// TwinCAT 3 PLC project xpp_pulsepicker_motion
// ProgramVersion: 3.1.4026.17
// libraries:
//   LCLS_OOPMotion, * (SLAC)
//   lcls_twincat_motion_synchronous, * (SLAC - LCLS)
//   PMPS, * (SLAC - LCLS)
//   Tc2_MC2, * (Beckhoff Automation GmbH)
//   Tc2_Standard, * (Beckhoff Automation GmbH)
//   Tc2_System, * (Beckhoff Automation GmbH)
//   TcUnit, * (www.tcunit.org)
// project tree:
//   DUTs/ E_ModeSelector.TcDUT, E_PickerState.TcDUT, E_StatusIndicator.TcDUT, E_ValidationStep.TcDUT, ST_SpeedProfile.TcDUT
//   / PlcTask.TcTTO
//   POUs/ FB_Burst.TcPOU, FB_FastClose.TcPOU, FB_FastOpen.TcPOU, FB_FlipFlop.TcPOU, FB_HomeToIndex.TcPOU, FB_MoveToNearestClosed.TcPOU, FB_OneShot.TcPOU, FB_PulsePicker.TcPOU, FB_SyncrhonousTest.TcPOU, MAIN.TcPOU
// real-time tasks:
//   TASK PlcTask: cycle T#1ms, priority 20, ADS port 350
// motion (NC):
//   TASK NC-Task 1 SAF: cycle T#1ms, priority 4, ADS port 501
//   TASK NC-Task 1 SVB: cycle T#10ms, priority 8, ADS port 511
//   AXIS Spindle (id 1)
//     General: UnitName=Degree
//     OtherSettings: AllowMotionCmdToSlave=true
//     encoder EncType=1
//     drive DrvType=5
//       Analog: TorqueSetpointScale=10, ScaleFactorActTorque=0.1
//       TimeComp: TaskDelayCycles=1
//     controller CtrType=1
//       CtrPara: PriorControlFactor=1
//         Observer: BandWidth=20
//   AXIS X (id 2)
//     OtherSettings: AllowMotionCmdToSlave=true
//     encoder EncType=1
//     drive DrvType=5
//       Analog: TorqueSetpointScale=10, ScaleFactorActTorque=0.1
//     controller CtrType=1
//       CtrPara: PriorControlFactor=1
//         Observer: BandWidth=20
//   AXIS Y (id 3)
//     OtherSettings: AllowMotionCmdToSlave=true
//     encoder EncType=1
//     drive DrvType=5
//       Analog: TorqueSetpointScale=10, ScaleFactorActTorque=0.1
//     controller CtrType=1
//       CtrPara: PriorControlFactor=1
//         Observer: BandWidth=20
// variable links:
//   xpp_pulsepicker_motion Instance <-> NC-Task 1 SAF/Axes/Spindle
//     PlcTask Inputs/MAIN.FB_SyncrhonousTest.AxisRef.NcToPlc <-> Outputs/ToPlc
//     PlcTask Outputs/MAIN.FB_SyncrhonousTest.AxisRef.PlcToNc <-> Inputs/FromPlc

CONFIGURATION xpp_pulsepicker_motion
    RESOURCE PLC ON TwinCAT3
        TASK PlcTask(INTERVAL := T#1ms, PRIORITY := 20);
        PROGRAM MAIN WITH PlcTask : MAIN;
    END_RESOURCE
END_CONFIGURATION

// ---- DUTs/E_ModeSelector.TcDUT
{attribute 'qualified_only'}
{attribute 'to_string'}
TYPE E_ModeSelector :
(
    ModeNone := 0,         // No mode / idle
    OneShot := 1,          // Mode 1
    FlipFlop := 2,         // Mode 2
    Burst := 3,            // Mode 3
    FastOpen := 4,         // Mode 4
    FastClose := 5,        // Mode 5
    Home := 7,             // Mode 7
    Reset := 99            // Reset
) UINT;
END_TYPE

// ---- DUTs/E_PickerState.TcDUT
{attribute 'qualified_only'}
{attribute 'strict'}
{attribute 'to_string'}
TYPE E_PickerState :
(
    Init,           // Startup: Read ModeSelect/SlitStatusFlag from NV
    HardReset,      // Hard reset initialization
    SoftReset,      // Soft reset/common block
    ModeSelect,     // Idle/waiting for user/command mode selection
    ModeExecute,    // Executing selected mode (One-Shot, Flip-Flop, etc)
    ErrorState      // Error or drift handling and recovery
);
END_TYPE

// ---- DUTs/E_StatusIndicator.TcDUT
{attribute 'qualified_only'}
{attribute 'strict'}
{attribute 'to_string'}
TYPE E_StatusIndicator :
(
// Mode Select/Resets
    WaitModeSelect := 0,
    // One-Shot
    OneShotInit := 10,
    OneShotLoopWait := 11,
    OneShotComplete := 12,
    // Flip-Flop
    FlipFlopInit := 20,
    FlipFlopLoopWait := 21,
    FlipFlopActive := 22,
    // Burst
    BurstInit := 30,
    BurstLoop := 31,
    // Fast Open/Close
    FastOpenInit := 40,
    FastOpenComplete := 41,
    FastCloseInit := 50,
    FastCloseComplete := 51,
    // Homing
    HomingInit := 70,
    HomingComplete := 79,
    // Special states
    HardReset := 80,
    SoftReset := 81
);
END_TYPE

// ---- DUTs/E_ValidationStep.TcDUT
{attribute 'qualified_only'}
{attribute 'strict'}
{attribute 'to_string'}
TYPE E_ValidationStep :
(
	INITIALIZE := 0,
	WAIT_FOR_IDLE,
	COMMAND_SEQUENCE_START,
	GENERATE_TARGET_POINTS,
	COMMAND_MOVE_TO_FIRST_TARGET,
	COMMAND_START_TRIGGERS,
	CONFIRM_BACK_TO_IDLE
);
END_TYPE

// ---- DUTs/ST_SpeedProfile.TcDUT
TYPE ST_SpeedProfile :
STRUCT
	InitialVelocity : LREAL;
	MaxVelocity : LREAL;
	Acceleration : LREAL;
	Deceleration : LREAL;
END_STRUCT
END_TYPE

// ---- POUs/MAIN.TcPOU
PROGRAM MAIN
VAR
	FB_SyncrhonousTest : FB_SyncrhonousTest;
END_VAR

FB_SyncrhonousTest();

END_PROGRAM

// ---- POUs/FB_SyncrhonousTest.TcPOU
FUNCTION_BLOCK FB_SyncrhonousTest
VAR
    (* --- Axis Reference --- *)
    AxisRef : AXIS_REF;

	fbPersistentDataStorage : FB_PersistentDataStorage;
    fbMotionStage : FB_MotionStageNC(
        sName := 'Test2',
         AxisRef := AxisRef,
        iPersistentDataStorage := fbPersistentDataStorage
    ) := (HomeMode:=E_EpicsHomeCmd.LOW_LIMIT);
	
    (* --- Timing, Trigger, and Clock --- *)
//     fbClockSourceInternal    : FB_ClockSourceInternal(
//         nTimePerScan := 250000,            // 0.25 ms cycle
//         nStartingTime := 0
//     );
    fbClockSourceInternal    : FB_ClockSourceInternal(
        nTimePerScan := 1000000,            // 1 ms cycle
        nStartingTime := 0
    );	
 	fbClockSourceEtherCATDistributedClock : FB_ClockSourceEtherCATDistributedClock;
//     fbTriggerSourceInternal : FB_TriggerSourceInternal(
//         iClockSource := fbClockSourceEtherCATDistributedClock
//     );
    fbTriggerSourceInternal : FB_TriggerSourceInternal(
        iClockSource := fbClockSourceEtherCATDistributedClock
    );
	
    fbTriggerManagerInternal : FB_TriggerManager(
        fTriggerFrequencyExpected := 30.0,  // 30 Hz expected trigger input
        iTriggerSource := fbTriggerSourceInternal
    );
//     fbTrajectoryClockSynchronous: FB_TrajectoryClockSynchronous (
//         fCycleTime := 0.000250,
//         iClockSource := fbClockSourceEtherCATDistributedClock
//     );
//     fbTrajectoryClockSynchronous: FB_TrajectoryClockSynchronous (
//         fCycleTime := 0.000250,
//         iClockSource := fbClockSourceInternal
//     );
    fbTrajectoryClockSynchronous: FB_TrajectoryClockSynchronous (
        fCycleTime := 0.001,
        iClockSource := fbClockSourceInternal
    );
    (* --- Trajectory and Buffer --- *)
    fbTargetPointSynchronousQueue        : FB_TargetPointSynchronousQueue<6>;   // Buffer of size 6
    fbTargetPointSynchronousLoader     		 : FB_TargetPointSynchronousLoaderFromEpics<1,6>(
        nMaxNumPointsProcessedPerCycle := 10
    );

    (* --- Setpoint & Feedback Interfaces --- *)
    fbSetpointInterfaceNC  : FB_SetpointInterfaceNC(AxisRef := AxisRef);
    fbFeedbackInterfaceNC  : FB_FeedbackInterfaceNC(AxisRef := AxisRef);

    (* --- Trajectory Synchronous and Error Estimation --- *)
    fbTrajectorySynchronous : FB_TrajectorySynchronousBezierContinuousSnap(
        iTrajectoryClock := fbTrajectoryClockSynchronous,
		bCalcPosPoints := TRUE,
		bCalcVelPoints := TRUE,
		bCalcAccPoints := TRUE,
		bCalcJerkPoints := TRUE,
		bCalcSnapPoints := TRUE
    );
    fbErrorEstimator     : FB_ErrorEstimator(
        iTrajectoryClock := fbTrajectoryClockSynchronous,
        iFeedbackInterface := fbFeedbackInterfaceNC,
        iTargetPointSynchronousQueue := fbTargetPointSynchronousQueue,
        iTrajectorySynchronous := fbTrajectorySynchronous,
        iTriggerManager := fbTriggerManagerInternal
    );

    (* --- Setpoint Generator --- *)
    fbSetpointGeneratorContinuousSynchronous : FB_SetpointGeneratorContinuousSynchronous(
        fTimeSyncGain := 0.2,
		iSetpointInterface := fbSetpointInterfaceNC,
		iFeedbackInterface := fbFeedbackInterfaceNC,
		iErrorEstimator := fbErrorEstimator,
		iTrajectorySynchronous := fbTrajectorySynchronous,
		iTargetPointSynchronousQueue := fbTargetPointSynchronousQueue,
		iTrajectoryClock := fbTrajectoryClockSynchronous,
		iTriggerManager := fbTriggerManagerInternal
    );

    (* --- Sequencer and EPICS Command/Loader --- *)
    fbTrajectorySequencerCommandsFromEpics : FB_TrajectorySequencerCommandsFromEpics;
	
    fbTrajectorySequencerSynchronous : FB_TrajectorySequencerSynchronous<1>(
        iTriggerManager := fbTriggerManagerInternal,
        iTrajectorySequencerCommands := fbTrajectorySequencerCommandsFromEpics
    );

	arTrajectoryPositions : ARRAY[1..6] OF LREAL := [
		-11.25,   // up: start
		-6.11,    // up: end / down: start
		-0.33,    // down: end / flat: start
		 0.33,    // flat: end / ramp2: start
		 6.12,    // ramp2: end / final: start
		11.25     // final: end
	];
	
	arTargetVelocities : ARRAY[1..6] OF LREAL := [
		 0.0,     // up: start
	  2400.0,     // up: end / down: start
	   300.0,     // down: end / flat: start
	   300.0,     // flat: end / ramp2: start
	  2400.0,     // ramp2: end / final: start
		 0.0      // final: end
	];
	
	arTargetTime : ARRAY[1..6] OF LREAL := [
	  0.0,            // up: start
	  0.0042828125,   // up: end / down: start
	  0.008565625,    // down: end / flat: start
	  0.010765625,    // flat: end / ramp2: start
	  0.0150484375,   // ramp2: end / final: start
	  0.01933125      // final: end
	];
    stPoint : ST_TrajectorySynchronousPoint;
	fbTargetPointSynchronous : FB_TargetPointSynchronous;
	bHardwareEnableSync AT %Q* :  BOOL;
	i : INT;
    (* --- Optionally: index/scan flags, and utility vars for test harness --- *)
    firstScan  : BOOL := TRUE;
    nIndex     : INT  := 1;         // Not needed for single axis, just in case
    seqStep    : E_TrajectorySequenceStep;
    isIdle     : BOOL;
	eUserState : E_ValidationStep;
	bHome: BOOL;
	bStartCommand: BOOL;
	bCommandMoveToFirstTarget: BOOL;
	bQuitEarly: BOOL;
	bStartTriggers: BOOL;
END_VAR

IF firstScan THEN

	bHardwareEnableSync := TRUE;
	fbMotionStage.EnableMode := LCLS_OOPMotion.E_StageEnableMode.ALWAYS;
	fbMotionStage.MotionCmd.nCmdData := LCLS_OOPMotion.E_EpicsHomeCmd.LOW_LIMIT;
	fbMotionStage.MotionCmd.fVelocity:=12.5;
	fbMotionStage.MotionCmd.fDeceleration := 25.5;
	fbMotionStage.MotionCmd.fAcceleration:=25.5;
	fbMotionStage.MotionCmd.fHomePosition := 0;

//     fbTriggerSource.Start(
//         fFrequency := 30.0,
//         nTotalNumTriggers := 1
//     );
// 	
//     fbTriggerSource.Reset();
//     fbTrajectorySequencerSynchronous.Register(
//         iTargetPointSynchronousQueue := fbTargetPointSynchronousQueue,
//         iSetpointGeneratorContinuous := fbSetpointGen,
//         iMotionStage := fbMotionStage,            // Use the motion axis FB here!
//         iSetpointInterface := fbSetpointInterface
//     );
    firstScan := FALSE;
END_IF

IF bHome THEN
	fbMotionStage.MotionCmd.bHomeCmd := TRUE;
	bHome := FALSE;
END_IF

fbClockSourceInternal();
//fbClockSourceEtherCATDistributedClock();
fbTriggerSourceInternal();
fbTrajectoryClockSynchronous();
fbTriggerManagerInternal();

// call for each axis
fbMotionStage();

fbSetpointInterfaceNC();
fbErrorEstimator();
fbSetpointGeneratorContinuousSynchronous();
fbTrajectorySequencerSynchronous();
///////////////////////////////////
fbTrajectorySequencerSynchronous();

CASE eUserState OF
	E_ValidationStep.INITIALIZE:
	 	fbTriggerSourceInternal.Reset();
        //fbTriggerManager.ResetTriggerCounter();
        fbTriggerManagerInternal.ResetTriggerCounter();
		
		fbTrajectorySequencerSynchronous.Register(
			iTargetPointSynchronousQueue := fbTargetPointSynchronousQueue,
			iSetpointGeneratorContinuous := fbSetpointGeneratorContinuousSynchronous,
			iMotionStage := fbMotionStage,            // Use the motion axis FB here!
			iSetpointInterface := fbSetpointInterfaceNC
		);
		eUserState := E_ValidationStep.WAIT_FOR_IDLE;
		
    E_ValidationStep.WAIT_FOR_IDLE:
        IF fbTrajectorySequencerSynchronous.eSequenceStep = E_TrajectorySequenceStep.IDLE THEN
            eUserState := E_ValidationStep.COMMAND_SEQUENCE_START;
        END_IF
		
    E_ValidationStep.COMMAND_SEQUENCE_START:
		IF bStartCommand THEN
			fbTrajectorySequencerCommandsFromEpics.CommandSequenceStart := TRUE;
		
			eUserState := E_ValidationStep.GENERATE_TARGET_POINTS;
			
			bStartCommand := FALSE;
		END_IF
	E_ValidationStep.GENERATE_TARGET_POINTS:
		FOR i := 1 TO 6 DO
			fbTargetPointSynchronous.Position := arTrajectoryPositions[i];
			fbTargetPointSynchronous.T := arTargetTime[i];
	
			fbTargetPointSynchronous.Velocity := arTargetVelocities[i];   // If your system uses velocity (optional)
			fbTargetPointSynchronous.Acceleration := 0.0;
			fbTargetPointSynchronous.Jerk := 0.0;
			fbTargetPointSynchronous.Snap := 0.0;
			fbTargetPointSynchronousQueue.Push(fbTargetPointSynchronous);
		END_FOR
		eUserState := E_ValidationStep.COMMAND_MOVE_TO_FIRST_TARGET;
		
    E_ValidationStep.COMMAND_MOVE_TO_FIRST_TARGET:
        IF bCommandMoveToFirstTarget THEN
            fbTrajectorySequencerCommandsFromEpics.CommandSequenceMoveToFirstTarget := TRUE;

            eUserState := E_ValidationStep.COMMAND_START_TRIGGERS;
			
			bCommandMoveToFirstTarget := FALSE;
        ELSIF fbTrajectorySequencerSynchronous.eSequenceStep = E_TrajectorySequenceStep.CONF_ERROR_RESET THEN
            bQuitEarly := TRUE;
        END_IF
		
    E_ValidationStep.COMMAND_START_TRIGGERS:
        IF bStartTriggers THEN
            //fbTriggerSourceInternal.Start(fFrequency := GVL_Constants.fTargetFrequency, nTotalNumTriggers := nNumTargets);
			fbTriggerSourceInternal.Start(
				fFrequency := 30.0,
				nTotalNumTriggers := 1
			);
            eUserState := E_ValidationStep.CONFIRM_BACK_TO_IDLE;
			
			bStartTriggers := FALSE;
        ELSIF fbTrajectorySequencerSynchronous.eSequenceStep = E_TrajectorySequenceStep.CONF_ERROR_RESET THEN
            bQuitEarly := TRUE;
        END_IF
		
	E_ValidationStep.CONFIRM_BACK_TO_IDLE:
        IF fbTrajectorySequencerSynchronous.eSequenceStep = E_TrajectorySequenceStep.IDLE THEN
            eUserState := E_ValidationStep.COMMAND_SEQUENCE_START;
        ELSIF fbTrajectorySequencerSynchronous.eSequenceStep = E_TrajectorySequenceStep.CONF_ERROR_RESET THEN
            bQuitEarly := TRUE;
        END_IF
END_CASE

END_FUNCTION_BLOCK

// ---- POUs/FB_Burst.TcPOU
FUNCTION_BLOCK FB_Burst
VAR_INPUT
    MotorCenterPosition : INT;              // P0
    MotorClosedPositionPlus : INT;          // P1
    EncoderCenterPosition : INT;            // N0
    EncoderClosedPositionPlus : INT;        // N1
    DriftLimit : INT;                       // Dl
    ErrorCheckEnabled : BOOL;               // Ec
    C2 : INT;                               // Actual encoder count
    InputTrip : BOOL;                       // Rising edge is Input trigger
END_VAR
VAR_IN_OUT
    EncoderShadow : INT;                    // Cs (shadow reg)
    SlitStatusFlag : INT;                   // Df
    UpperDriftViolations : INT;             // Ud
    LowerDriftViolations : INT;             // Ld
END_VAR
VAR_OUTPUT
    Complete : BOOL := FALSE;               // Set TRUE when any move is complete
END_VAR
VAR
    State : INT := 0;                       // 0=idle, 1=open move, 2=close move, 10=waiting for input
    Drift : INT := 0;
    InputTripLast : BOOL := FALSE;          // For edge detection
END_VAR

METHOD Execute
// Edge detection
VAR
    Trip : BOOL;
END_VAR
Trip := InputTrip AND NOT InputTripLast;
InputTripLast := InputTrip;

// Main burst loop. User triggers with input pulse.
// Initial state: waiting for InputTrip, Df determines direction
IF State = 0 THEN
    IF Trip THEN
        IF SlitStatusFlag = 1 THEN     // Currently closed, need to open on trip
            StartOpenMove();
        ELSE                           // Currently open, need to close on trip
            StartCloseMove();
        END_IF
    END_IF
ELSIF State = 1 THEN
    // J3: Burst Open ISR
    // Move shutter to open position (MotorCenterPosition)
    // Replace with MC_MoveAbsolute or actual axis block (simulate instant success here)
    IF ErrorCheckEnabled AND (SlitStatusFlag = 1) THEN
        Drift := EncoderClosedPositionPlus - EncoderShadow; // N1-Cs
        IF Drift >= DriftLimit THEN
            LowerDriftViolations := LowerDriftViolations + 1;
        END_IF
    END_IF
    EncoderShadow := C2;
    SlitStatusFlag := 0;   // Slits are open
    State := 10;           // Waiting for next input pulse
    Complete := TRUE;

ELSIF State = 2 THEN
    // J4: Burst Close ISR
    // Move shutter to closed position (MotorClosedPositionPlus)
    // Replace with MC_MoveAbsolute or actual axis block (simulate instant success here)
    IF ErrorCheckEnabled THEN
        Drift := EncoderShadow - EncoderCenterPosition; // Cs-N0
        IF Drift >= DriftLimit THEN
            UpperDriftViolations := UpperDriftViolations + 1;
        END_IF
    END_IF
    EncoderShadow := C2;
    SlitStatusFlag := 1;   // Slits are closed
    State := 10;           // Waiting for next input pulse
    Complete := TRUE;

ELSIF State = 10 THEN
    // Await next trigger
    IF Trip THEN
        IF SlitStatusFlag = 1 THEN
            StartOpenMove();
        ELSE
            StartCloseMove();
        END_IF
    END_IF
END_IF
END_METHOD

METHOD StartCloseMove
VAR_INPUT
END_VAR
    State := 2;          // Start close move ISR (J4)
    Complete := FALSE;
END_METHOD

METHOD StartOpenMove
VAR_INPUT
END_VAR
    State := 1;          // Start open move ISR (J3)
    Complete := FALSE;
END_METHOD

END_FUNCTION_BLOCK

// ---- POUs/FB_FastClose.TcPOU
FUNCTION_BLOCK FB_FastClose
VAR_INPUT
    MotorClosedPositionPlus : INT;       // P1 (positive closed)
    C2 : INT;                            // Encoder actual count
    SlitStatusFlagIn : INT;              // Input Df for position check
END_VAR
VAR_IN_OUT
    EncoderShadow : INT;                 // Cs (shadow register)
    SlitStatusFlag : INT;                // Df
END_VAR
VAR_OUTPUT
    Complete : BOOL := FALSE;
END_VAR
VAR
    State : INT := 0; // 0: idle, 1: moving, 2: done
END_VAR

METHOD Execute : BOOL
VAR_INPUT
END_VAR
IF State = 0 THEN
    // Only move if not already closed
    IF (SlitStatusFlagIn <> 1) AND (SlitStatusFlagIn <> -1) THEN
        State := 1;       // Start moving to P1
        Complete := FALSE;
    ELSE
        // Already closed, skip to complete
        State := 2;
        Complete := TRUE;
    END_IF
ELSIF State = 1 THEN
    // Simulate motion complete; check actual axis in a real system
    EncoderShadow := C2;
    SlitStatusFlag := 1;   // Positive closed
    State := 2;
    Complete := TRUE;
END_IF
END_METHOD

METHOD Reset : BOOL
VAR_INPUT
END_VAR
    State := 0;
    Complete := FALSE;
END_METHOD

END_FUNCTION_BLOCK

// ---- POUs/FB_FastOpen.TcPOU
FUNCTION_BLOCK  FB_FastOpen
VAR_INPUT
    MotorCenterPosition : INT;           // P0 (open pos)
    C2 : INT;                            // Encoder actual count
END_VAR
VAR_IN_OUT
    EncoderShadow : INT;                 // Cs (shadow register)
    SlitStatusFlag : INT;                // Df
END_VAR
VAR_OUTPUT
    Complete : BOOL := FALSE;
END_VAR
VAR
    State : INT := 0; // 0: idle, 1: moving, 2: done
END_VAR

METHOD Execute : BOOL
VAR_INPUT
END_VAR
IF State = 0 THEN
    // Start movement to open (simulate instant success; call MC_MoveAbsolute in real system)
    State := 1;
    Complete := FALSE;
ELSIF State = 1 THEN
    // Simulate motion complete; check actual motion in real system
    EncoderShadow := C2;
    SlitStatusFlag := 0;      // Open
    State := 2;
    Complete := TRUE;
END_IF
END_METHOD

METHOD Reset : BOOL
VAR_INPUT
END_VAR
    State := 0;
    Complete := FALSE;
END_METHOD

END_FUNCTION_BLOCK

// ---- POUs/FB_FlipFlop.TcPOU
FUNCTION_BLOCK FB_FlipFlop
VAR_INPUT
    MotorClosedPositionPlus  : INT;            // P1
    MotorClosedPositionMinus : INT;            // P2
    EncoderClosedPositionPlus: INT;            // N1
    EncoderClosedPositionMinus: INT;           // N2
    DriftLimit               : INT;
    ErrorCheckEnabled        : BOOL;
    C2                       : INT;            // encoder count
    InputTrip                : BOOL;           // TRUE on input pulse
END_VAR
VAR_IN_OUT
    EncoderShadow            : INT;            // Cs
    SlitStatusFlag           : INT;            // Df
    UpperDriftViolations     : INT;            // Ud
    LowerDriftViolations     : INT;            // Ld
END_VAR
VAR_OUTPUT
    Complete                 : BOOL := FALSE;  // TRUE when first move done
END_VAR
VAR
    NextDirectionPos         : BOOL := TRUE;   // TRUE: Arm ISR2/J6, FALSE: Arm ISR1/J5
    State                    : INT := 0;       // 0: idle/init; 1: closed pos armed; 2: waiting trip; 3: actuation/move
    LastInputTrip            : BOOL := FALSE;  // For edge detection
    Drift                    : INT := 0;
END_VAR

METHOD Execute : BOOL
VAR
    Trip : BOOL;
END_VAR
Trip := InputTrip AND NOT LastInputTrip;
LastInputTrip := InputTrip;

// Init: ensure we're at positive or negative closed
IF State=0 THEN
    IF (SlitStatusFlag = -1) THEN
        NextDirectionPos := TRUE;  // Arm ISR2/J6 on trip
    ELSE
        NextDirectionPos := FALSE; // Arm ISR1/J5 on trip
    END_IF
    State := 1;
    Complete := TRUE;              // First move is done on entry
ELSIF State=1 OR State=2 THEN
    // Wait for input trip
    IF Trip THEN
        State := 3;
        Complete := FALSE;
    END_IF
ELSIF State=3 THEN
    // Do move and drift calculation
    IF NextDirectionPos THEN
        // ISR2/J6: P2→P1
        // Move motor to P1 (simulate instant for demo)
        IF ErrorCheckEnabled THEN
            Drift := EncoderShadow - EncoderClosedPositionMinus; // Cs-N2
            IF Drift >= DriftLimit THEN
                UpperDriftViolations := UpperDriftViolations + 1;
            END_IF
        END_IF
        SlitStatusFlag := 1;    // Positive closed
        EncoderShadow := C2;
        NextDirectionPos := FALSE; // Next trip arms negative direction (J5)
    ELSE
        // ISR1/J5: P1→P2
        // Move motor to P2 (simulate instant for demo)
        IF ErrorCheckEnabled THEN
            Drift := EncoderClosedPositionPlus - EncoderShadow; // N1-Cs
            IF Drift >= DriftLimit THEN
                LowerDriftViolations := LowerDriftViolations + 1;
            END_IF
        END_IF
        SlitStatusFlag := -1;   // Negative closed
        EncoderShadow := C2;
        NextDirectionPos := TRUE; // Next trip arms positive direction (J6)
    END_IF
    State := 2;    // Return to wait for input trip
    Complete := TRUE;
END_IF
END_METHOD

METHOD Reset : BOOL
VAR_INPUT
END_VAR
    State := 0;
    Complete := FALSE;
    NextDirectionPos := TRUE; // Default to J6
END_METHOD

END_FUNCTION_BLOCK

// ---- POUs/FB_HomeToIndex.TcPOU
FUNCTION_BLOCK FB_HomeToIndex
VAR_INPUT
    MotorClosedPositionPlus : INT;   // P1
    EncoderClosedPositionPlus: INT;  // N1
    MagicOffset : INT;               // Mo
    HomingSpeed : LREAL;      // CL V9 (see earlier struct)
    VM : LREAL;                        // Max velocity (from speed profile)
END_VAR
VAR_IN_OUT
    EncoderShadow : INT;             // Cs
    SlitStatusFlag : INT;            // Df
    Ud : INT;                        // Upper drift violation counter
    Lowerd : INT;                        // Lower drift violation counter
END_VAR
VAR_OUTPUT
    Complete : BOOL := FALSE;
END_VAR
VAR
    State : INT := 0;
    DoneHome : BOOL := FALSE;
    DoneOffset : BOOL := FALSE;
END_VAR

METHOD Execute : BOOL
VAR_INPUT
END_VAR
// State 0: Start Homing
IF State = 0 THEN
    // Load homing speed profile (CL V9) - can set to axis FB
    // (Your MC_Home or similar FB called here with VM etc.)
    // For demo, just set DoneHome true immediately, replace with real move!
    DoneHome := TRUE;
    State := 1;
END_IF

// State 1: Wait for Homing move complete
IF State = 1 THEN
    IF DoneHome THEN
        // Now do relative move by magic offset to positive closed (P1)
        // MC_MoveRelative(Mo ...) here in real system!
        DoneOffset := TRUE;
        State := 2;
    END_IF
END_IF

// State 2: Wait for move by Mo complete
IF State = 2 THEN
    IF DoneOffset THEN
        // Set C1 and C2 appropriately
        // In real code, set axis reference to MotorClosedPositionPlus
        // Set encoder reference to EncoderClosedPositionPlus
        // Sync shadow register
        // Set slit state Df to known positive closed
        SlitStatusFlag := 1;
        EncoderShadow := EncoderClosedPositionPlus;
        Ud := 0;
        Lowerd := 0;
        Complete := TRUE;
        State := 3;
    END_IF
END_IF
END_METHOD

METHOD Reset : BOOL
VAR_INPUT
END_VAR
    State := 0;
    DoneHome := FALSE;
    DoneOffset := FALSE;
    Complete := FALSE;
END_METHOD

END_FUNCTION_BLOCK

// ---- POUs/FB_MoveToNearestClosed.TcPOU
FUNCTION_BLOCK FB_MoveToNearestClosed
VAR_INPUT
    MotorClosedPositionPlus : INT;    // P1
    C2 : INT;                         // Actual encoder count (from axis/encoder)
    SlitStatusFlagIn : INT;           // Input Df (current position status)
END_VAR
VAR_IN_OUT
    EncoderShadow : INT;              // Cs, shadow register for drift checking
    SlitStatusFlag : INT;             // Df, output position status
END_VAR
VAR_OUTPUT
    Complete : BOOL := FALSE;
END_VAR
VAR
    State : INT := 0;                 // 0: ready, 1: moving, 2: done
END_VAR

METHOD Execute : BOOL
VAR_INPUT
END_VAR
IF State = 0 THEN
    IF (SlitStatusFlagIn <> 1) AND (SlitStatusFlagIn <> -1) THEN
        // Start the move to P1 (simulate or call MC_MoveAbsolute)
        State := 1;
        Complete := FALSE;
    ELSE
        // Already closed; nothing to do
        State := 2;
        Complete := TRUE;
    END_IF
ELSIF State = 1 THEN
    // Simulate move complete; in real code, check axis feedback!
    EncoderShadow := C2;
    SlitStatusFlag := 1;         // Signal at positive closed position
    State := 2;
    Complete := TRUE;
END_IF
END_METHOD

METHOD Reset : BOOL
VAR_INPUT
END_VAR
    State := 0;
    Complete := FALSE;
END_METHOD

END_FUNCTION_BLOCK

// ---- POUs/FB_OneShot.TcPOU
FUNCTION_BLOCK FB_OneShot
VAR_INPUT
    MotorClosedPositionPlus : INT;        // P1
    MotorClosedPositionMinus : INT;       // P2
    EncoderClosedPositionPlus : INT;      // N1
    EncoderClosedPositionMinus : INT;     // N2
    DriftLimit : INT;                     // Dl
    ErrorCheckEnabled : BOOL;             // Ec
    C2 : INT;                             // Actual encoder count
    ArmDirectionPos : BOOL := TRUE;       // TRUE: arm ISR2/P2→P1, FALSE: arm ISR1/P1→P2
    TriggerInputTrip : BOOL;              // TRUE when Input Trip triggers the action
END_VAR
VAR_IN_OUT
    EncoderShadow : INT;                  // Cs
    SlitStatusFlag : INT;                 // Df
    UpperDriftViolations : INT;           // Ud
    LowerDriftViolations : INT;           // Ld
END_VAR
VAR_OUTPUT
    Complete : BOOL := FALSE;             // Set TRUE when done
END_VAR
VAR
    Drift : INT := 0;
    MotionState : INT := 0;               // 0: idle/armed, 1: running, 2: done
END_VAR

METHOD Execute : BOOL
VAR_INPUT
END_VAR
// Call cyclically while armed; runs the ISR sequence after Input Trip
IF MotionState = 0 THEN
    // Nothing until InputTrip triggers
    IF TriggerInputTrip THEN
        MotionState := 1;         // Begin movement
        Complete := FALSE;
    END_IF
ELSIF MotionState = 1 THEN
    // Axis move (simulate or use your axis FB)
    IF ArmDirectionPos THEN
        // Move P2=>P1 (positive)
        // Example: AxisControl.MoveAbs(MotorClosedPositionPlus) -- Replace with FB or IO
        // Simulate motion complete immediately for demo!
        IF ErrorCheckEnabled THEN
            Drift := EncoderShadow - EncoderClosedPositionMinus; // Dr = Cs - N2
            IF Drift >= DriftLimit THEN
                UpperDriftViolations := UpperDriftViolations + 1;
            END_IF
        END_IF
        SlitStatusFlag := 1;     // Positive closed
    ELSE
        // Move P1=>P2 (negative)
        // Example: AxisControl.MoveAbs(MotorClosedPositionMinus)
        IF ErrorCheckEnabled THEN
            Drift := EncoderClosedPositionPlus - EncoderShadow; // Dr = N1 - Cs
            IF Drift >= DriftLimit THEN
                LowerDriftViolations := LowerDriftViolations + 1;
            END_IF
        END_IF
        SlitStatusFlag := -1;    // Negative closed
    END_IF
    EncoderShadow := C2;
    MotionState := 2;             // Finished
    Complete := TRUE;
END_IF
END_METHOD

METHOD Reset : BOOL
VAR_INPUT
END_VAR
    MotionState := 0;
    Complete := FALSE;
END_METHOD

END_FUNCTION_BLOCK

// ---- POUs/FB_PulsePicker.TcPOU
FUNCTION_BLOCK FB_PulsePicker
VAR PERSISTENT
    ModeSelect : E_ModeSelector := E_ModeSelector.ModeNone;;
 	StatusIndicator : E_StatusIndicator := E_StatusIndicator.WaitModeSelect;
    SlitStatusFlag : INT := 99;
    SweepDistance : INT;      
    EncoderSweepDistance : INT;
    EncoderDrift : INT;
    DriftLimit : INT;
    MotorCenterPosition : INT;
    MotorClosedPositionPlus : INT;    // P1
    MotorClosedPositionMinus : INT;   // P2
    EncoderCenterPosition : INT;      // N0
    EncoderClosedPositionPlus : INT;  // N1
    EncoderClosedPositionMinus : INT; // N2
    ErrorCheckEnabled : BOOL;
    MCodeVersion : INT;
    HeartbeatCounter : INT;
    EncoderShadow : INT;              // Cs
    UpperDriftViolations : INT;       // Ud
    LowerDriftViolations : INT;       // Ld
    HomingOffset : INT;               // Mo

END_VAR

VAR
    CurrentState : E_PickerState := E_PickerState.Init;
    ErrorCode : INT := 0;
    UserModeReq : UINT := 0;       // From HMI or remote
    (* Axis/encoder for simulation *)
    C2 : INT := 0;                // Encoder actual count from axis/IO
    (* Axis/encoder for simulation *)


    (* Speed profiles *)
    V1_Speed : ST_SpeedProfile := (InitialVelocity := 7500, MaxVelocity := 10000, Acceleration := 1875000, Deceleration := 1875000);
    V2_Speed : ST_SpeedProfile := (InitialVelocity := 7500, MaxVelocity := 10000, Acceleration := 1875000, Deceleration := 1875000);
    V3_Speed : ST_SpeedProfile := (InitialVelocity := 5300, MaxVelocity := 10000, Acceleration := 1875000, Deceleration := 1875000);
    V4_Speed : ST_SpeedProfile := (InitialVelocity := 5300, MaxVelocity := 10000, Acceleration := 1875000, Deceleration := 1875000);
    V5_Speed : ST_SpeedProfile := (InitialVelocity := 5300, MaxVelocity := 10000, Acceleration := 1875000, Deceleration := 1875000);
    V9_Speed : ST_SpeedProfile := (InitialVelocity := 640,   MaxVelocity := 2560,  Acceleration := 640,    Deceleration := 640);

    (* FB instances *)
    fbMoveToNearestClosed : FB_MoveToNearestClosed;
    fbOneShot : FB_OneShot;
    fbBurst   : FB_Burst;
    fbFlipFlop: FB_FlipFlop;
    fbFastOpen: FB_FastOpen;
    fbFastClose: FB_FastClose;
    fbHomeToIndex: FB_HomeToIndex;

    (* Flags/input trips *)
    OneShotInputTrip : BOOL := FALSE;
    OneShotActive : BOOL := FALSE;
    OneShotDirectionPos : BOOL := TRUE;

    BurstInputTrip : BOOL := FALSE;
    BurstInitDone : BOOL := FALSE;

    FlipFlopInputTrip : BOOL := FALSE;
    FlipFlopInitDone : BOOL := FALSE;

    FastOpenInitDone : BOOL := FALSE;
    FastCloseInitDone : BOOL := FALSE;
    HomingInitDone : BOOL := FALSE;

    ActiveSpeedProfile : ST_SpeedProfile;
END_VAR

(* =========================
   Main State Machine Logic
   ========================= *)
CASE CurrentState OF

    E_PickerState.Init:
        IF ModeSelect <> E_ModeSelector.ModeNone THEN
            StatusIndicator := E_StatusIndicator.HardReset;           // Hard Reset Init
            ModeSelect := E_ModeSelector.Reset;
            SlitStatusFlag := 99;
            CurrentState := E_PickerState.HardReset;
        ELSE
            StatusIndicator := E_StatusIndicator.SoftReset;           // Soft Reset Init
            ModeSelect := E_ModeSelector.ModeNone;
            CurrentState := E_PickerState.SoftReset;
        END_IF

    E_PickerState.HardReset:
        StatusIndicator := E_StatusIndicator.HardReset;
        ModeSelect := E_ModeSelector.Reset;
        SlitStatusFlag := 99;
        StatusIndicator := E_StatusIndicator.SoftReset;               // Go to soft reset next
        CurrentState := E_PickerState.SoftReset;

    E_PickerState.SoftReset:
        StatusIndicator := E_StatusIndicator.SoftReset;
        HeartbeatCounter := 0;
        ModeSelect := E_ModeSelector.ModeNone;
        CurrentState := E_PickerState.ModeSelect;

    E_PickerState.ModeSelect:
        StatusIndicator := E_StatusIndicator.WaitModeSelect;
        HeartbeatCounter := HeartbeatCounter + 1;

        IF SlitStatusFlag = 99 THEN
            ErrorCode := 1;
            StatusIndicator := E_StatusIndicator.HardReset;
            CurrentState := E_PickerState.ErrorState;
        ELSIF ErrorCode <> 0 THEN
            CurrentState := E_PickerState.ErrorState;
        ELSIF (UserModeReq >= E_ModeSelector.OneShot) AND (UserModeReq <= E_ModeSelector.Home) THEN
            ModeSelect := UserModeReq;
            CurrentState := E_PickerState.ModeExecute;
        END_IF

    E_PickerState.ModeExecute:
        CASE ModeSelect OF
        
            E_ModeSelector.OneShot:
                CASE StatusIndicator OF
                    E_StatusIndicator.WaitModeSelect, E_StatusIndicator.OneShotInit:
                        StatusIndicator := E_StatusIndicator.OneShotInit;
                        ActiveSpeedProfile := V1_Speed;

                        // ... (the rest is unchanged, just update status codes) ...

                        StatusIndicator := E_StatusIndicator.OneShotLoopWait;

                    E_StatusIndicator.OneShotLoopWait:
                        HeartbeatCounter := HeartbeatCounter + 1;
                        fbOneShot.TriggerInputTrip := OneShotActive AND OneShotInputTrip;
                        fbOneShot.Execute();

                        // ...
                        IF ModeSelect = E_ModeSelector.ModeNone THEN
                            StatusIndicator := E_StatusIndicator.WaitModeSelect;
                            CurrentState := E_PickerState.ModeSelect;
                        ELSIF ModeSelect = E_ModeSelector.FastClose THEN
                            StatusIndicator := E_StatusIndicator.FastCloseInit;
                            CurrentState := E_PickerState.ModeExecute;
                        END_IF
                END_CASE

            E_ModeSelector.FlipFlop:
                CASE StatusIndicator OF
                    E_StatusIndicator.WaitModeSelect, E_StatusIndicator.FlipFlopInit:
                        StatusIndicator := E_StatusIndicator.FlipFlopInit;
                        ActiveSpeedProfile := V2_Speed;
                        IF NOT FlipFlopInitDone THEN
                            // ...
                            FlipFlopInitDone := TRUE;
                        END_IF
                        // ...
                        IF fbMoveToNearestClosed.Complete THEN
                            // ...
                            StatusIndicator := E_StatusIndicator.FlipFlopLoopWait;
                            FlipFlopInitDone := FALSE;
                        END_IF
                    E_StatusIndicator.FlipFlopLoopWait:
                        HeartbeatCounter := HeartbeatCounter + 1;
                        fbFlipFlop.Execute();
                        // ...
                        IF ModeSelect = E_ModeSelector.ModeNone THEN
                            StatusIndicator := E_StatusIndicator.WaitModeSelect;
                            CurrentState := E_PickerState.ModeSelect;
                        ELSIF ModeSelect = E_ModeSelector.FastClose THEN
                            StatusIndicator := E_StatusIndicator.FastCloseInit;
                            CurrentState := E_PickerState.ModeExecute;
                        END_IF
                END_CASE

            E_ModeSelector.Burst:
                CASE StatusIndicator OF
                    E_StatusIndicator.WaitModeSelect, E_StatusIndicator.BurstInit:
                        StatusIndicator := E_StatusIndicator.BurstInit;
                        ActiveSpeedProfile := V3_Speed;
                        IF NOT BurstInitDone THEN
                            // ...
                            BurstInitDone := TRUE;
                        END_IF
                        // ...
                        IF fbMoveToNearestClosed.Complete THEN
                            // ...
                            BurstInitDone := FALSE;
                            StatusIndicator := E_StatusIndicator.BurstLoop;
                        END_IF
                    E_StatusIndicator.BurstLoop:
                        HeartbeatCounter := HeartbeatCounter + 1;
                        fbBurst.Execute();
                        // ...
                        IF ModeSelect = E_ModeSelector.ModeNone THEN
                            StatusIndicator := E_StatusIndicator.WaitModeSelect;
                            CurrentState := E_PickerState.ModeSelect;
                        ELSIF ModeSelect = E_ModeSelector.FastClose THEN
                            StatusIndicator := E_StatusIndicator.FastCloseInit;
                            CurrentState := E_PickerState.ModeExecute;
                        END_IF
                END_CASE

            E_ModeSelector.FastOpen:
                CASE StatusIndicator OF
                    E_StatusIndicator.WaitModeSelect, E_StatusIndicator.FastOpenInit:
                        StatusIndicator := E_StatusIndicator.FastOpenInit;
                        ActiveSpeedProfile := V4_Speed;
                        fbFastOpen.Reset();
                        fbFastOpen.MotorCenterPosition := MotorCenterPosition;
                        fbFastOpen.C2 := C2;
                        fbFastOpen.EncoderShadow := EncoderShadow;
                        fbFastOpen.SlitStatusFlag := SlitStatusFlag;
                        StatusIndicator := E_StatusIndicator.FastOpenComplete;
                    E_StatusIndicator.FastOpenComplete:
                        fbFastOpen.Execute();
                        EncoderShadow := fbFastOpen.EncoderShadow;
                        SlitStatusFlag := fbFastOpen.SlitStatusFlag;
                        IF fbFastOpen.Complete THEN
                            ModeSelect := E_ModeSelector.ModeNone;
                            CurrentState := E_PickerState.ModeSelect;
                        END_IF
                END_CASE

            E_ModeSelector.FastClose:
                CASE StatusIndicator OF
                    E_StatusIndicator.WaitModeSelect, E_StatusIndicator.FastCloseInit:
                        StatusIndicator := E_StatusIndicator.FastCloseInit;
                        ActiveSpeedProfile := V5_Speed;
                        fbFastClose.Reset();
                        fbFastClose.MotorClosedPositionPlus := MotorClosedPositionPlus;
                        fbFastClose.C2 := C2;
                        fbFastClose.EncoderShadow := EncoderShadow;
                        fbFastClose.SlitStatusFlag := SlitStatusFlag;
                        fbFastClose.SlitStatusFlagIn := SlitStatusFlag;
                        StatusIndicator := E_StatusIndicator.FastCloseComplete;
                    E_StatusIndicator.FastCloseComplete:
                        fbFastClose.Execute();
                        EncoderShadow := fbFastClose.EncoderShadow;
                        SlitStatusFlag := fbFastClose.SlitStatusFlag;
                        IF fbFastClose.Complete THEN
                            ModeSelect := E_ModeSelector.ModeNone;
                            CurrentState := E_PickerState.ModeSelect;
                        END_IF
                END_CASE

            E_ModeSelector.Home:
                CASE StatusIndicator OF
                    E_StatusIndicator.WaitModeSelect, E_StatusIndicator.HomingInit:
                        StatusIndicator := E_StatusIndicator.HomingInit;
                        ActiveSpeedProfile := V9_Speed;
                        IF NOT HomingInitDone THEN
                            fbHomeToIndex.Reset();
                            fbHomeToIndex.MotorClosedPositionPlus := MotorClosedPositionPlus;
                            fbHomeToIndex.EncoderClosedPositionPlus := EncoderClosedPositionPlus;
                            fbHomeToIndex.MagicOffset := HomingOffset;
                            fbHomeToIndex.HomingSpeed := V9_Speed;
                            fbHomeToIndex.VM := V9_Speed.MaxVelocity;
                            fbHomeToIndex.EncoderShadow := EncoderShadow;
                            fbHomeToIndex.SlitStatusFlag := SlitStatusFlag;
                            fbHomeToIndex.Ud := UpperDriftViolations;
                            fbHomeToIndex.Lowerd := LowerDriftViolations;
                            HomingInitDone := TRUE;
                        END_IF
                        fbHomeToIndex.Execute();
                        EncoderShadow := fbHomeToIndex.EncoderShadow;
                        SlitStatusFlag := fbHomeToIndex.SlitStatusFlag;
                        UpperDriftViolations := fbHomeToIndex.Ud;
                        LowerDriftViolations := fbHomeToIndex.Ld;
                        IF fbHomeToIndex.Complete THEN
                            HomingInitDone := FALSE;
                            StatusIndicator := E_StatusIndicator.HomingComplete;
                            ModeSelect := E_ModeSelector.ModeNone;
                            CurrentState := E_PickerState.ModeSelect;
                        END_IF
                END_CASE
            ELSE
                StatusIndicator := E_StatusIndicator.WaitModeSelect;
                ModeSelect := E_ModeSelector.ModeNone;
                CurrentState := E_PickerState.ModeSelect;
        END_CASE

    E_PickerState.ErrorState:
        IF (SlitStatusFlag = 99) AND (UserModeReq = E_ModeSelector.Home) THEN
            StatusIndicator := E_StatusIndicator.HomingInit;
            fbHomeToIndex.Reset();
            fbHomeToIndex.MotorClosedPositionPlus := MotorClosedPositionPlus;
            fbHomeToIndex.EncoderClosedPositionPlus := EncoderClosedPositionPlus;
            fbHomeToIndex.MagicOffset := HomingOffset;
            fbHomeToIndex.HomingSpeed := V9_Speed;
            fbHomeToIndex.VM := V9_Speed.MaxVelocity;
            fbHomeToIndex.EncoderShadow := EncoderShadow;
            fbHomeToIndex.SlitStatusFlag := SlitStatusFlag;
            fbHomeToIndex.Ud := UpperDriftViolations;
            fbHomeToIndex.Lowerd := LowerDriftViolations;
            fbHomeToIndex.Execute();
            EncoderShadow := fbHomeToIndex.EncoderShadow;
            SlitStatusFlag := fbHomeToIndex.SlitStatusFlag;
            UpperDriftViolations := fbHomeToIndex.Ud;
            LowerDriftViolations := fbHomeToIndex.Lowerd;
            IF fbHomeToIndex.Complete THEN
                StatusIndicator := E_StatusIndicator.HomingComplete;
                ErrorCode := 0;
                ModeSelect := E_ModeSelector.ModeNone;
                CurrentState := E_PickerState.ModeSelect;
            END_IF
        END_IF

    ELSE
        CurrentState := E_PickerState.Init;

END_CASE

END_FUNCTION_BLOCK
